// TIA Portal V17 export
// export: Created 2022-07-28T18:03:21.8821686Z, ExportSetting None, DisplayName Totally Integrated Automation Portal, DisplayVersion V17, DisplayName TIA Portal Openness, DisplayVersion V17, DisplayName TIA Portal Teamcenter Gateway, DisplayVersion V17, DisplayName TIA Portal Version Control Interface, DisplayVersion V17, DisplayName TIA Portal Test Suite Advanced, DisplayVersion V17, DisplayName SINAMICS Startdrive Advanced, DisplayVersion V17, DisplayName SINAMICS DCC, DisplayVersion V17, DisplayName SINAMICS Startdrive G130, G150, S120, S150, SINAMICS MV, S210, DisplayVersion V17, DisplayName SINAMICS Startdrive G110M, G120, G120C, G120D, G120P, G115D, DisplayVersion V17, DisplayName STEP 7 Professional, DisplayVersion V17, DisplayName SIMATIC Energy Suite, DisplayVersion V17, DisplayName STEP 7 CFC, DisplayVersion V17, DisplayName STEP 7 Safety, DisplayVersion V17, DisplayName WinCC Advanced / Unified PC, DisplayVersion V17, DisplayName SIMATIC Visualization Architect, DisplayVersion V17
TYPE "_SlideGate_Blow_Config"
   STRUCT
      "b" { ExternalAccessible := 'False'; ExternalVisible := 'False'; ExternalWritable := 'False'} : Struct   // bool parameters
         AutoAskErrors { S7_SetPoint := 'True'} : Bool;
         AutoResetInterlock { S7_SetPoint := 'True'} : Bool;
         SimAutoSensorChange { S7_SetPoint := 'True'} : Bool;   // Start autocalibrate process
         bit_3 { S7_SetPoint := 'True'} : Bool := true;   // Enable auto change sensor state in simulation mode
         bit_4 { S7_SetPoint := 'True'} : Bool;   // Open/close by time r_TimeWalk
         bit_5 { S7_SetPoint := 'True'} : Bool;
         bit_6 { S7_SetPoint := 'True'} : Bool;
         bit_7 { S7_SetPoint := 'True'} : Bool;
      END_STRUCT;
      r_SP_TimePause : Real := 120.0;   // Set point of time for pause, s
      r_SP_TimeWork : Real := 5.0;   // Set point of time for work, s
      r_PV_LeftTime { ExternalWritable := 'False'} : Real := 0.0;   // Left time to work, s
      w_enableExternalErrors_16 { ExternalAccessible := 'False'; ExternalVisible := 'False'; ExternalWritable := 'False'; S7_SetPoint := 'True'} : Word := 16#FFFF;   // bit - 1 = enable
      b_bypassInterlocksForward_8 { ExternalAccessible := 'False'; ExternalVisible := 'False'; ExternalWritable := 'False'; S7_SetPoint := 'True'} : Byte := 16#FF;   // bit - 0 = Interlock Bypassed forward direction
      b_bypassInterlocksReverse_8 { ExternalAccessible := 'False'; ExternalVisible := 'False'; ExternalWritable := 'False'; S7_SetPoint := 'True'} : Byte := 16#FF;   // bit - 0 = Interlock Bypassed reverse direction
   END_STRUCT;
END_TYPE
